{attribute 'GeneratedUsingTerminal: EP9224-0037-0017'}
{attribute addProperty BoxType "EP9224-0037-0017"}
{attribute addProperty Id "A_0022_EP9224_0037_0017_2_EP9224_1037EP9224_1FC0878B2"}
{attribute addProperty CRC "3458496376"}
{attribute addProperty Size "2"}
TYPE A_0022_EP9224_0037_0017_CE247778 EXTENDS EP9224_079410B7 :
STRUCT
	{attribute addProperty Name "A_0022_EP9224_0037_0017_2_EP9224_1037"}
	{attribute addProperty PreviousPort "A_0022(EP9224-0037-0017) : D"}
	A_0022_EP9224_0037_0017_2_EP9224_1037 : EP9224_1FC0878B;
END_STRUCT
END_TYPE

(* stored: Version 1.2.0.0, ProductVersion 3.1.4024.9
   DUT A_0022_EP9224_0037_0017_CE247778: Id {00d39572-1746-4178-9122-c00989829079} *)
